// Mitsubishi GX Developer project: D-2-1   PLC: FX2N

PROGRAM Main
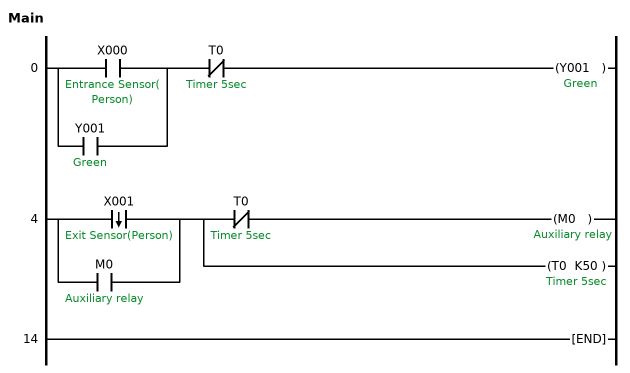
0     LD      X000  ; Entrance Sensor(Person)
      OR      Y001  ; Green
      ANI     T0  ; Timer 5sec
      OUT     Y001  ; Green
4     LDF     X001  ; Exit Sensor(Person)
      OR      M0  ; Auxiliary relay
      MPS
      ANI     T0  ; Timer 5sec
      OUT     M0  ; Auxiliary relay
      MPP
      OUT     T0 K50  ; Timer 5sec
14    END
END_PROGRAM
